(* Logix 5000 project; controller EsteiraSeletoraParte1 vendor 1 type 14 code 89 rev 20.11; software revision 20.05 *)

TASK MainTask (continuous, watchdog 500 ms) : MainProgram

MODULES
   Controller : vendor 1 type 14 code 89 (CompactLogixL23E_QBFC1_Controller 0, rev 20.11)
      LocalENB : vendor 1 type 12 code 191 (CompactLogixL23E_QBFC1_Ethernet 1, rev 20.11)
      Local : CompactBus (CompactVirtualAdapter 3, rev 20.11)
         Discrete_Inputs : vendor 1 type 7 code 320 (Compact 1, rev 3.1, Input RPI 20 ms)
         Discrete_Outputs : vendor 1 type 7 code 322 (Compact 2, rev 3.1, Output RPI 20 ms)
         Analog_IO : vendor 1 type 10 code 120 (Compact 3, rev 1.1, Output RPI 80 ms)
         Counters : vendor 1 type 109 code 70 (Compact 4, rev 1.1, Output RPI 20 ms)
END_MODULES

PROGRAM MainProgram   (* main routine MainRoutine *)
VAR
   AcionaPistao : ALIAS FOR Local:2:O.Data.8;
   EsperaMetal : TIMER;
   EsperaNaoMetal : TIMER;
   EsperaPistao : TIMER;
   PassandoMetal : BOOL;
   PassandoNaoMetal : BOOL;
   SensorIndutivo : ALIAS FOR Local:1:I.Data.8;
   SensorLuz : ALIAS FOR Local:1:I.Data.9;
   SensorPresenca : BOOL;
   SistemaLigado : BOOL;
   StartStop : ALIAS FOR Local:1:I.Data.3;
END_VAR

ROUTINE MainRoutine   (* ladder *)
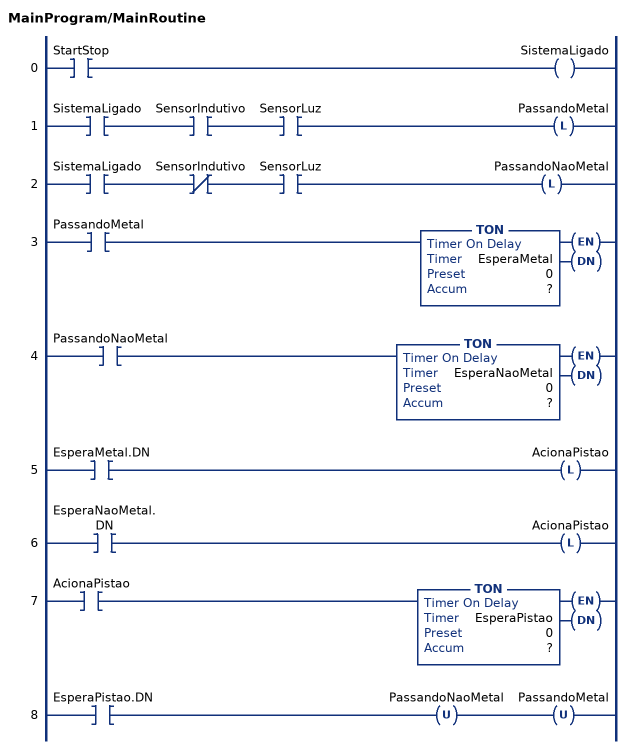
   0: XIC(StartStop)OTE(SistemaLigado);
   1: XIC(SistemaLigado)XIC(SensorIndutivo)XIC(SensorLuz)OTL(PassandoMetal);
   2: XIC(SistemaLigado)XIO(SensorIndutivo)XIC(SensorLuz)OTL(PassandoNaoMetal);
   3: XIC(PassandoMetal)TON(EsperaMetal,?,?);
   4: XIC(PassandoNaoMetal)TON(EsperaNaoMetal,?,?);
   5: XIC(EsperaMetal.DN)OTL(AcionaPistao);
   6: XIC(EsperaNaoMetal.DN)OTL(AcionaPistao);
   7: XIC(AcionaPistao)TON(EsperaPistao,?,?);
   8: XIC(EsperaPistao.DN)OTU(PassandoNaoMetal)OTU(PassandoMetal);
END_ROUTINE
END_PROGRAM
